// TIA Portal V20 export
TYPE "LKinCtrl_typePoint"
   STRUCT
      "name" : WString["LKINCTRL_LENGTH_OF_CMDPOINT_NAME"];   // Specification of a point name
      position : Array[0..5] of LReal;   // Specification of Cartesian position for a point
      coordSystem : USInt;   // Specification of a point coordinate system
      linkConstellation : DWord := 16#FFFF_FFFF;   // Specification of the target link constellation
      turnJoint : Array[0..5] of DInt;   // Only relevant with more than four interpolating kinematics axes - When "CoordSystem" = 0, 1, 2 or 3: target joint position range of the joint J[1..6]
   END_STRUCT;
END_TYPE
